(* IEC 61131-3 sources: volt/packages/volt-lsp-iec/test-corpus/pro2193/Device/Plc Logic/Application/09 Misc/Library Manager/SysExcept, 3 files *)

(* ---- REGCONTEXT.dut ---- *)
TYPE REGCONTEXT :
STRUCT
	IP : __UXINT;
	BP : __UXINT;
	SP : __UXINT;
END_STRUCT
END_TYPE

(* ---- RTSEXCEPTIONS.gvl ---- *)
VAR_GLOBAL
	RTSEXCPT_UNKNOWN : UDINT := SINT_TO_UDINT(-1);
	RTSEXCPT_NOEXCEPTION : UDINT := 16#0;
	RTSEXCPT_WATCHDOG : UDINT := 16#10;
	RTSEXCPT_HARDWAREWATCHDOG : UDINT := 16#11;
	RTSEXCPT_IO_CONFIG_ERROR : UDINT := 16#12;
	RTSEXCPT_PROGRAMCHECKSUM : UDINT := 16#13;
	RTSEXCPT_FIELDBUS_ERROR : UDINT := 16#14;
	RTSEXCPT_IOUPDATE_ERROR : UDINT := 16#15;
	RTSEXCPT_CYCLE_TIME_EXCEED : UDINT := 16#16;
	RTSEXCPT_ONLCHANGE_PROGRAM_EXCEEDED : UDINT := 16#17;
	RTSEXCPT_UNRESOLVED_EXTREFS : UDINT := 16#18;
	RTSEXCPT_DOWNLOAD_REJECTED : UDINT := 16#19;
	RTSEXCPT_BOOTPROJECT_REJECTED_DUE_RETAIN_ERROR : UDINT := 16#1A;
	RTSEXCPT_LOADBOOTPROJECT_FAILED : UDINT := 16#1B;
	RTSEXCPT_OUT_OF_MEMORY : UDINT := 16#1C;
	RTSEXCPT_RETAIN_MEMORY_ERROR : UDINT := 16#1D;
	RTSEXCPT_BOOTPROJECT_CRASH : UDINT := 16#1E;
	RTSEXCPT_BOOTPROJECTTARGETMISMATCH : UDINT := 16#21;
	RTSEXCPT_SCHEDULEERROR : UDINT := 16#22;
	RTSEXCPT_FILE_CHECKSUM_ERR : UDINT := 16#23;
	RTSEXCPT_RETAIN_IDENTITY_MISMATCH : UDINT := 16#24;
	RTSEXCPT_IEC_TASK_CONFIG_ERROR : UDINT := 16#25;
	RTSEXCPT_APP_TARGET_MISMATCH : UDINT := 16#26;
	RTSEXCPT_ILLEGAL_INSTRUCTION : UDINT := 16#50;
	RTSEXCPT_ACCESS_VIOLATION : UDINT := 16#51;
	RTSEXCPT_PRIV_INSTRUCTION : UDINT := 16#52;
	RTSEXCPT_IN_PAGE_ERROR : UDINT := 16#53;
	RTSEXCPT_STACK_OVERFLOW : UDINT := 16#54;
	RTSEXCPT_INVALID_DISPOSITION : UDINT := 16#55;
	RTSEXCPT_INVALID_HANDLE : UDINT := 16#56;
	RTSEXCPT_GUARD_PAGE : UDINT := 16#57;
	RTSEXCPT_DOUBLE_FAULT : UDINT := 16#58;
	RTSEXCPT_INVALID_OPCODE : UDINT := 16#59;
	RTSEXCPT_MISALIGNMENT : UDINT := 16#100;
	RTSEXCPT_ARRAYBOUNDS : UDINT := 16#101;
	RTSEXCPT_DIVIDEBYZERO : UDINT := 16#102;
	RTSEXCPT_OVERFLOW : UDINT := 16#103;
	RTSEXCPT_NONCONTINUABLE : UDINT := 16#104;
	RTSEXCPT_PROCESSORLOAD_WATCHDOG : UDINT := 16#105;
	RTSEXCPT_FPU_ERROR : UDINT := 16#150;
	RTSEXCPT_FPU_DENORMAL_OPERAND : UDINT := 16#151;
	RTSEXCPT_FPU_DIVIDEBYZERO : UDINT := 16#152;
	RTSEXCPT_FPU_INEXACT_RESULT : UDINT := 16#153;
	RTSEXCPT_FPU_INVALID_OPERATION : UDINT := 16#154;
	RTSEXCPT_FPU_OVERFLOW : UDINT := 16#155;
	RTSEXCPT_FPU_STACK_CHECK : UDINT := 16#156;
	RTSEXCPT_FPU_UNDERFLOW : UDINT := 16#157;
	RTSEXCPT_VENDOR_EXCEPTION_BASE : UDINT := 16#2000;
END_VAR

(* ---- SYSEXCEPTGENERATEEXCEPTION.pou ---- *)
FUNCTION SYSEXCEPTGENERATEEXCEPTION : RTS_IEC_RESULT
VAR_INPUT
	UDIEXCEPTION : UDINT;
END_VAR
END_FUNCTION
